TYPE ST_AC_Siemens :
STRUCT
	Protocol: STRING;
	Model : STRING;
END_STRUCT
END_TYPE

(* stored: Version 1.1.0.1, ProductVersion 3.1.4024.9
   DUT ST_AC_Siemens: Id {5d06c8a0-5e90-42f1-a0e8-d1f1bc027d80} *)
